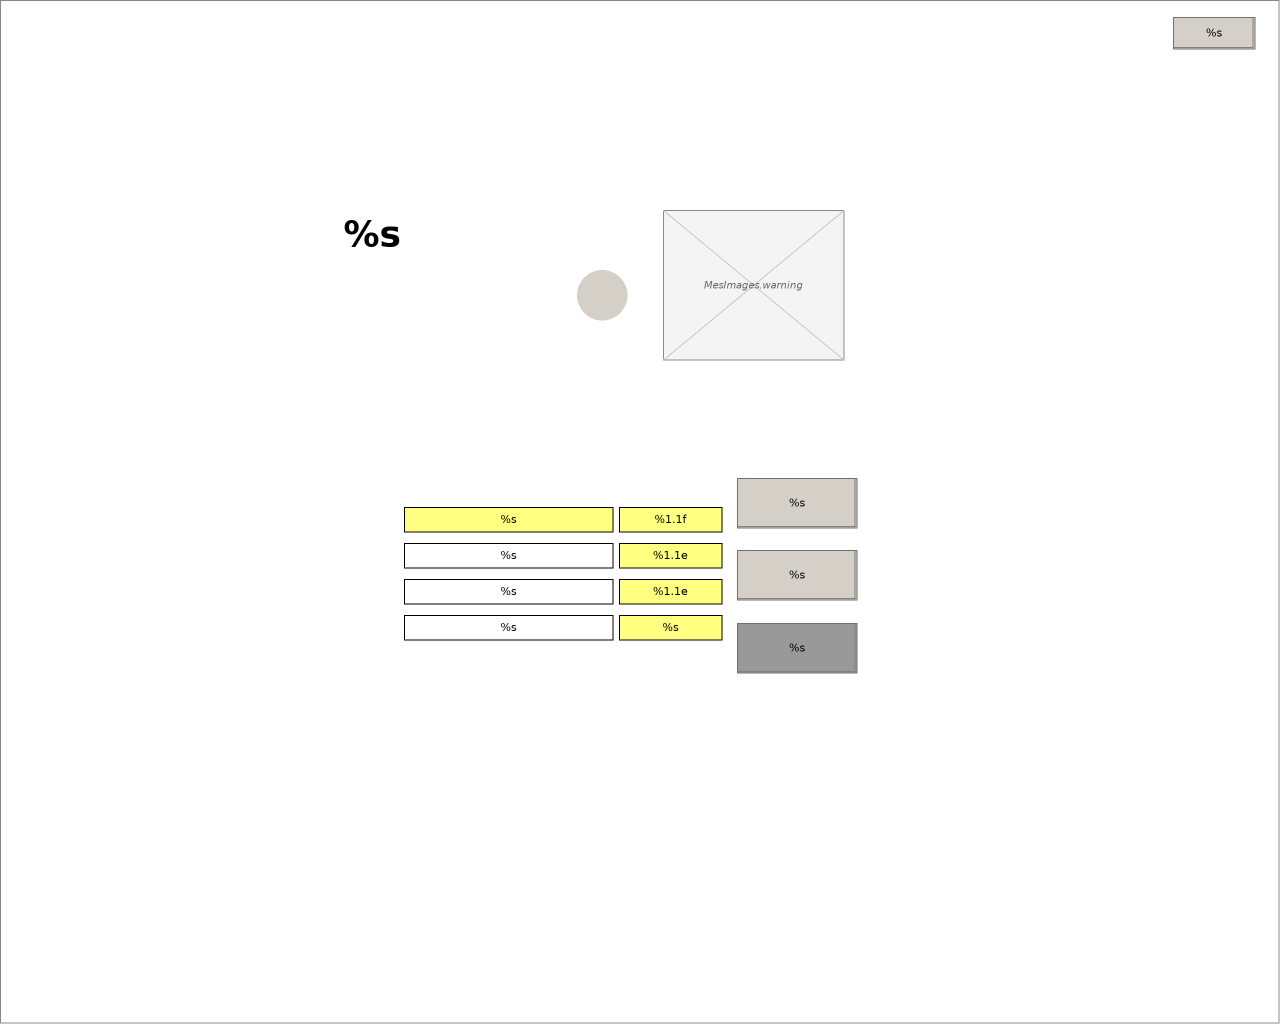
VISUALIZATION VISU_VANNE_ASS_VAT653_ETHERCAT_MANU  // 1280x1024
VAR_IN_OUT
	m_Input_Vanne:		BLOCK_VVAT_653_ETHERCAT;
	m_Input_State_Manu:	BOOL;
END_VAR
    Button (1173,17 82x32), "%s", text list: 'TextList_Basiques', text index: 8
        OnMouseClick: change screen: Previous 
        OnMouseClick: execute { .VISU_INDEX_MANU := 0; }
    Polygon (0,0), colour toggle: m_Input_VANNE.STATE_Lam
    Rectangle (290,200 165x68), "%s", text variable: m_Input_VANNE.MNEMO
    Polygon (0,0), colour toggle: m_Input_VANNE.STATE_On, invisible if: NOT (m_Input_VANNE.STATE_Off OR m_Input_VANNE.STATE_On)
    Ellipse (577,270 50x50), colour toggle: m_Input_VANNE.STATE_Ok, invisible if: NOT m_Input_VANNE.STATE_Ok
    Image (663,210 181x150), invisible if: NOT m_Input_VANNE.STATE_Nok, image: MesImages.warning
    Button (737,478 120x50), "%s", input disabled if: NOT m_Input_Vanne.AUTOR_On_IHM OR NOT .PRG_USER.ACTU_USER.MAINTENANCE, text list: 'TextList_VVAT_3P', text index: 0
        toggle m_Input_Vanne.M_On
    Button (737,550 120x50), "%s", input disabled if: NOT m_Input_Vanne.AUTOR_Off_IHM OR NOT .PRG_USER.ACTU_USER.MAINTENANCE, text list: 'TextList_VVAT_3P', text index: 1
        toggle m_Input_Vanne.M_Off
    Button (737,623 120x50), "%s", input disabled if: NOT m_Input_Vanne.AUTOR_Lam_IHM OR NOT .PRG_USER.ACTU_USER.MAINTENANCE, text list: 'TextList_VVAT_3P', text index: 2
        toggle m_Input_Vanne.M_Lam
    RoundedRectangle (404,507 209x25), "%s", invisible if: NOT m_Input_Vanne.PRM_Mode, input disabled if: NOT .PRG_USER.ACTU_USER.MAINTENANCE OR NOT m_Input_State_Manu OR NOT m_Input_Vanne.PRM_Mode, text list: 'TextList_VVAT_650_ETHERCAT', text index: 8
        OnMouseClick: toggle m_Input_Vanne.PRM_Mode
    RoundedRectangle (404,507 209x25), "%s", invisible if: m_Input_Vanne.PRM_Mode, input disabled if: NOT .PRG_USER.ACTU_USER.MAINTENANCE OR NOT m_Input_State_Manu OR m_Input_Vanne.PRM_Mode, text list: 'TextList_VVAT_650_ETHERCAT', text index: 7
        OnMouseClick: toggle m_Input_Vanne.PRM_Mode
    RoundedRectangle (404,543 209x25), "%s", invisible if: NOT m_Input_Vanne.PRM_Mode, text list: 'TextList_VVAT_650_ETHERCAT', text index: 4
    RoundedRectangle (404,579 209x25), "%s", invisible if: NOT m_Input_Vanne.PRM_Mode, text list: 'TextList_VVAT_650_ETHERCAT', text index: 5
    RoundedRectangle (404,615 209x25), "%s", invisible if: NOT m_Input_Vanne.PRM_Mode, text list: 'TextList_VVAT_650_ETHERCAT', text index: 6
    RoundedRectangle (619,615 103x25), "%s", text variable: m_Input_Vanne.PRM_Tim_W_Pr, invisible if: NOT m_Input_Vanne.PRM_Mode, input disabled if: NOT m_Input_Vanne.PRM_Mode
        OnMouseClick: write the text variable via VisuDialogs.Keypad
    RoundedRectangle (619,579 103x25), "%1.1e", text variable: m_Input_Vanne.PRM_W_Pr_HI, invisible if: NOT m_Input_Vanne.PRM_Mode, input disabled if: NOT m_Input_Vanne.PRM_Mode
        OnMouseClick: write the text variable via VisuDialogs.NumpadExtended, min 0, max 1000
    RoundedRectangle (619,543 103x25), "%1.1e", text variable: m_Input_Vanne.PRM_W_Pr_LO, invisible if: NOT m_Input_Vanne.PRM_Mode, input disabled if: NOT m_Input_Vanne.PRM_Mode
        OnMouseClick: write the text variable via VisuDialogs.NumpadExtended, min 0, max 1000
    RoundedRectangle (619,507 103x25), "%1.1e", text variable: m_Input_Vanne.PRM_Pression, invisible if: NOT m_Input_Vanne.PRM_Mode, input disabled if: NOT m_Input_Vanne.PRM_Mode
        OnMouseClick: write the text variable via VisuDialogs.NumpadExtended, min 0, max 1000
    RoundedRectangle (619,507 103x25), "%1.1f", text variable: m_Input_Vanne.PRM_Position, invisible if: m_Input_Vanne.PRM_Mode, input disabled if: m_Input_Vanne.PRM_Mode
        OnMouseClick: write the text variable via VisuDialogs.Numpad, min 0, max 100
END_VISUALIZATION

(* stored: Version 1.1.0.1, ProductVersion 3.1.4024.12
   Visu VISU_VANNE_ASS_VAT653_ETHERCAT_MANU: Id {a79a9b07-8404-4e23-8380-7d05bf7e3122} *)
